//---------------------------------------------------------------------------------------------------------------
//
//  HAUD 2026.04.10.
//
//  fb_XmlBase
//    - wraps xml read
//    - wraps xml write
//
//   - abstract base class for extending xml R/W ctrl for any data
//
//---------------------------------------------------------------------------------------------------------------
// This SOFTWARE is provided as an Example by THE PROVIDER "as is" and "with all faults." THE PROVIDER makes no 
// representations or warranties of any kind concerning the safety, suitability, lack of viruses, inaccuracies, 
// typographical errors, or other harmful components of this SOFTWARE. There are inherent dangers in the use of 
// any software, and you are solely responsible for determining whether this SOFTWARE is compatible with your 
// equipment and other software installed on your equipment. You are also solely responsible for the protection 
// of your equipment and backup of your data, and THE PROVIDER will not be liable for any damages you may suffer 
// in connection with using, modifying, or distributing this SOFTWARE.
//---------------------------------------------------------------------------------------------------------------
FUNCTION_BLOCK ABSTRACT fb_XmlBase
VAR
  //------------------------------------------------------------------------------------------------------------
  // pointer check result
  //------------------------------------------------------------------------------------------------------------
  _eCheck                     : E_DATA_CHECK;
  _sCheck                     : STRING;
  //------------------------------------------------------------------------------------------------------------
  // internal control and state
  //------------------------------------------------------------------------------------------------------------
  _eInit                      : E_PROGRESS;
  _eCmd,
  _eCmdOld                    : E_DATA_CTRL;
  _eState                     : E_DATA_STATE;
  _eResult                    : E_PROGRESS;
  //------------------------------------------------------------------------------------------------------------
  // Tc2_XmlDataSrv wrappers
  //------------------------------------------------------------------------------------------------------------
  _fbXmlRead                  : fb_XmlRead;
  _fbXmlWrite                 : fb_XmlWrite;
  //------------------------------------------------------------------------------------------------------------
  // who am I?
  //  - Identity built in extending class
  //
  // see fb_Configuration.Identity.Set() as example
  //------------------------------------------------------------------------------------------------------------
  {attribute 'displaymode' := 'hex'}
  _XpuIdentity                : OTCID;        // identity must be set by extending class
  _sIdentity                  : STRING;       // part of filename
  //------------------------------------------------------------------------------------------------------------
  // where am I?
  //  - hocus pocus
  //    - you have to define my locus 
  //
  // see fb_Configuration.Identity.Set() as example
  //------------------------------------------------------------------------------------------------------------
  _sDirectoryPath             : STRING;       // root directory for data
  _sFilePath                  : STRING(255);  // path and filename (shall include identity in filepath)

  _sName                      : STRING;       // filename with *.xml
  _sXpath                     : STRING;       // XPath from extending class
  //------------------------------------------------------------------------------------------------------------
  // what am I?
  //  - data from the void
  //------------------------------------------------------------------------------------------------------------
  _pData                      : Global.PVOID;
  _nData                      : UDINT;
  //------------------------------------------------------------------------------------------------------------
  _eDeviceIdentifier          : e_Device;
  _stMsg                      : ST_Message;
  _eMessageLevel              : E_MessageType;
END_VAR

METHOD CreateFolder : E_PROGRESS
VAR_INPUT
  Execute         : BOOL;
END_VAR
VAR_INST
  _nErrorId       : UDINT;
  _eState         : E_PROGRESS;
  _sPath          : Tc2_System.T_MaxString;
  _fbCreateDir    : Tc2_System.FB_CreateDir;
END_VAR

IF NOT Execute
THEN
  _eState                     := E_PROGRESS.PROGRESS_INIT;
END_IF


CASE _eState
OF
  E_PROGRESS.PROGRESS_INIT:
    IF Execute
    THEN
      _eState                 := E_PROGRESS.PROGRESS_BUSY;
      _nErrorId               := 0;

      _fbCreateDir(
                    sNetId    := '', 
                    sPathName := _sPath, 
                    ePath     := Tc2_System.E_OpenPath.PATH_GENERIC, 
                    bExecute  := FALSE, 
                    tTimeout  := T#1S);
    END_IF

  E_PROGRESS.PROGRESS_BUSY:
    _fbCreateDir(
                  sNetId      := '', 
                  sPathName   := _sPath, 
                  ePath       := Tc2_System.E_OpenPath.PATH_GENERIC, 
                  bExecute    := TRUE, 
                  tTimeout    := T#1S,
                  nErrId      => _nErrorId);

    IF _fbCreateDir.bBusy
    THEN
      _eState                 := E_PROGRESS.PROGRESS_OCCUPIED;
    END_IF

  E_PROGRESS.PROGRESS_OCCUPIED:
    _fbCreateDir(
                  sNetId      := '', 
                  sPathName   := _sPath, 
                  ePath       := Tc2_System.E_OpenPath.PATH_GENERIC, 
                  bExecute    := TRUE, 
                  tTimeout    := T#1S,
                  nErrId      => _nErrorId);

    IF NOT _fbCreateDir.bBusy
    THEN
      _eState                 := E_PROGRESS.PROGRESS_WORKING;
    END_IF

  E_PROGRESS.PROGRESS_WORKING:
    _eState                   := E_PROGRESS.PROGRESS_DONE;
    _fbCreateDir(
                  sNetId      := '', 
                  sPathName   := _sPath, 
                  ePath       := Tc2_System.E_OpenPath.PATH_GENERIC, 
                  bExecute    := FALSE, 
                  tTimeout    := T#1S);

    IF (_eMessageLevel > E_MessageType.eMessageError)
    THEN
      _stMsg.eType            := E_MessageType.eMessageInfo;
      _stMsg.eDevice          := _eDeviceIdentifier;
      _stMsg.eSubdevice       := e_Subdevice.fbCreateFolder;
      _stMsg.iErrorNumber     := 0;
      _stMsg.sText            := concat(' : ', TO_STRING(_eState));
      f_MessageSet(_stMsg);
    END_IF
END_CASE

CreateFolder                  := _eState;
END_METHOD

PROPERTY FilePath : string(255)
GET
FilePath := _sFilePath;
END_GET
END_PROPERTY

PROPERTY FolderPath : string
GET
FolderPath := _sDirectoryPath;
END_GET
SET
_sDirectoryPath := FolderPath;
END_SET
END_PROPERTY

PROPERTY MessageDevice : udint
SET
_eDeviceIdentifier   := MessageDevice;
END_SET
END_PROPERTY

PROPERTY MessageLevel : e_messagetype
SET
_eMessageLevel := MessageLevel;
END_SET
END_PROPERTY

METHOD XmlRead  : E_PROGRESS
VAR_INPUT
  Execute               : BOOL;
END_VAR
VAR_INST
  _eState               : E_PROGRESS;
  _nErrorId             : UDINT;
END_VAR

IF NOT Execute
THEN
  _eState                     := E_PROGRESS.PROGRESS_INIT;
END_IF

CASE _eState
OF
  E_PROGRESS.PROGRESS_INIT:
    IF Execute
    THEN
      _nErrorId               := 0;
      _eState                 := E_PROGRESS.PROGRESS_BUSY;

      IF (_eMessageLevel > E_MessageType.eMessageInfo)
      THEN
        _stMsg.eType          := E_MessageType.eMessageVerbose;
        _stMsg.eDevice        := _eDeviceIdentifier;
        _stMsg.eSubdevice     := e_Subdevice.fbXmlRead;
        _stMsg.iErrorNumber   := _nErrorId;
        _stMsg.sText          := concat(' : ', TO_STRING(_eState));
        f_MessageSet(_stMsg);
      END_IF
    END_IF

  E_PROGRESS.PROGRESS_BUSY:
    _eState                   := E_PROGRESS.PROGRESS_OCCUPIED;
    _fbXmlRead(
              bExecute        := FALSE, 
              sFilePath       := _sFilePath, 
              sXPath          := _sXpath, 
              pData           := _pData, 
              diSize          := _nData);

  E_PROGRESS.PROGRESS_OCCUPIED:
    _fbXmlRead(
              bExecute        := TRUE);

    IF _fbXmlRead.bError
    THEN
      _nErrorId               := _fbXmlRead.nError;
      _eState                 := E_PROGRESS.PROGRESS_ERROR;

      _stMsg.eType            := E_MessageType.eMessageError;
      _stMsg.eDevice          := _eDeviceIdentifier;
      _stMsg.eSubdevice       := e_Subdevice.fbXmlRead;
      _stMsg.iErrorNumber     := _nErrorId;
      _stMsg.sText            := concat(' : ', TO_STRING(_eState));
      f_MessageSet(_stMsg);

      _fbXmlRead(
              bExecute        := FALSE);

    ELSIF _fbXmlRead.bDone
    THEN
      _eState                 := E_PROGRESS.PROGRESS_WORKING;
      _fbXmlRead(
              bExecute        := FALSE);
    END_IF

  E_PROGRESS.PROGRESS_WORKING:
    _eState                   := E_PROGRESS.PROGRESS_DONE;

    IF (_eMessageLevel > E_MessageType.eMessageError)
    THEN
      _stMsg.eType            := E_MessageType.eMessageInfo;
      _stMsg.eDevice          := _eDeviceIdentifier;
      _stMsg.eSubdevice       := e_Subdevice.fbXmlRead;
      _stMsg.iErrorNumber     := _nErrorId;
      _stMsg.sText            := concat(' : ', TO_STRING(_eState));
      f_MessageSet(_stMsg);
    END_IF
END_CASE

XmlRead                       := _eState;
END_METHOD

METHOD XmlWrite : E_PROGRESS
VAR_INPUT
  Execute               : BOOL;
END_VAR
VAR_INST
  _eState               : E_PROGRESS;
  _nErrorId             : UDINT;
END_VAR

IF NOT Execute
THEN
  _eState                     := E_PROGRESS.PROGRESS_INIT;
END_IF

CASE _eState
OF
  E_PROGRESS.PROGRESS_INIT:
    IF Execute
    THEN
      _nErrorId               := 0;
      _eState                 := E_PROGRESS.PROGRESS_BUSY;

      IF (_eMessageLevel > E_MessageType.eMessageInfo)
      THEN
        _stMsg.eType          := E_MessageType.eMessageVerbose;
        _stMsg.eDevice        := _eDeviceIdentifier;
        _stMsg.eSubdevice     := e_Subdevice.fbXmlWrite;
        _stMsg.iErrorNumber   := _nErrorId;
        _stMsg.sText          := concat(' : ', TO_STRING(_eState));
        f_MessageSet(_stMsg);
      END_IF
    END_IF

  E_PROGRESS.PROGRESS_BUSY:
    _eState                   := E_PROGRESS.PROGRESS_OCCUPIED;
    _fbXmlWrite(
              bExecute        := FALSE, 
              sFilePath       := _sFilePath, 
              sXPath          := _sXpath, 
              pData           := _pData, 
              diSize          := _nData);

  E_PROGRESS.PROGRESS_OCCUPIED:
    _fbXmlWrite(
              bExecute        := TRUE);

    IF _fbXmlWrite.bError
    THEN
      _nErrorId               := _fbXmlRead.nError;
      _eState                 := E_PROGRESS.PROGRESS_ERROR;

      _stMsg.eType            := E_MessageType.eMessageError;
      _stMsg.eDevice          := _eDeviceIdentifier;
      _stMsg.eSubdevice       := e_Subdevice.fbXmlWrite;
      _stMsg.iErrorNumber     := _nErrorId;
      _stMsg.sText            := concat(' : ', TO_STRING(_eState));
      f_MessageSet(_stMsg);

      _fbXmlWrite(
              bExecute        := FALSE);

    ELSIF _fbXmlWrite.bDone
    THEN
      _eState                 := E_PROGRESS.PROGRESS_WORKING;
      _fbXmlWrite(
              bExecute        := FALSE);
    END_IF

  E_PROGRESS.PROGRESS_WORKING:
    _eState                   := E_PROGRESS.PROGRESS_DONE;

    IF (_eMessageLevel > E_MessageType.eMessageError)
    THEN
      _stMsg.eType            := E_MessageType.eMessageInfo;
      _stMsg.eDevice          := _eDeviceIdentifier;
      _stMsg.eSubdevice       := e_Subdevice.fbXmlWrite;
      _stMsg.iErrorNumber     := _nErrorId;
      _stMsg.sText            := concat(' : ', TO_STRING(_eState));
      f_MessageSet(_stMsg);
    END_IF
END_CASE

XmlWrite                      := _eState;
END_METHOD

END_FUNCTION_BLOCK

(* stored: Version 1.1.0.1
   POU fb_XmlBase: Id {782075df-f4e4-4da3-8365-d247d6d73979}, SpecialFunc None
   Folder methods: Id {2c89a67c-ccf2-41d3-b2da-70628f248897}
   Folder properties: Id {970b89e4-dcbe-48c6-9a65-2e59844f6c1f}
   Method CreateFolder: Id {cb8dc966-e83e-4e45-9d72-4357d9ed6b38}
   Property FilePath: Id {58c39793-6dbc-4513-b5ba-62ea538c84f0}
   Get Get: Id {ff52ddd8-0278-415f-b941-2ab8379f2dc6}
   Property FolderPath: Id {ca5d0d86-3266-4632-b593-7505dd54aebd}
   Get Get: Id {02fc648a-b92f-4b3e-8a98-3480514c4ecb}
   Set Set: Id {f90ebd16-68a2-49ce-ba4a-65f5a2bd1fd0}
   Property MessageDevice: Id {8df2a424-895e-458f-a578-233842a90430}
   Set Set: Id {cd542040-b4de-42a8-bf65-00d2a359e6d1}
   Property MessageLevel: Id {9ea3c4c9-0708-4846-9c05-4dee836dffa0}
   Set Set: Id {e3dbea5c-7dc3-4d33-8d0f-ba25733b22fa}
   Method XmlRead: Id {4637618d-754f-4cb5-a04c-1f56f6fe19c5}
   Method XmlWrite: Id {511ced58-5e03-4146-bf4f-539b2af3ae98} *)
